// TIA Portal V19 export
FUNCTION "Flow_Counter" : Void   // FC2, STL
{ S7_Optimized_Access := 'TRUE' }
// Product Flow Count - Side stream route to Hamba2/Gasti
// stored: AutoNumber false
BEGIN

NETWORK
TITLE = 
// reset count at CIP
      A     "TANK CLEAN";
      JCN   M001;
      L     0;
      T     "Flow Count".Prod_Vol_Count;

//check for pulse and increment count
M001: A     "M_AHV_STERILE";
      A     "M_Product_Available";
      A     "M_Product_Route";  //side stream barrier open
      A     "Pulse_ FT01.83";

      FP    "Flow_Pulse_Mem";
      A     "Flow_Pulse_Mem";
      JCN   M002;
      L     "Flow Count".Prod_Vol_Count;
      L     10.0;
      +R;


      T     "Flow Count".Prod_Vol_Count;






M002: A     "M_AHV_STERILE";
      A     "M_Product_Available";
      A     "M_Product_Route";
      =     "Tag_49";
      NOP   0;
END_FUNCTION
